TYPE DUT_Control_Base :
STRUCT
	Open :BOOL;
	Close :BOOL;
	Reset :BOOL;
	Simulation :BOOL;
	AutoOn :BOOL;
	AutoOff :BOOL;
	ManualOn :BOOL;
	ManualOff :BOOL;
END_STRUCT
END_TYPE

(* stored: Version 1.1.0.1, ProductVersion 3.1.4024.12
   DUT DUT_Control_Base: Id {e2a918e7-e4ea-455c-969c-2b8567061d2f} *)
